Universal Robots PolyScope program: var_counter_106.urp

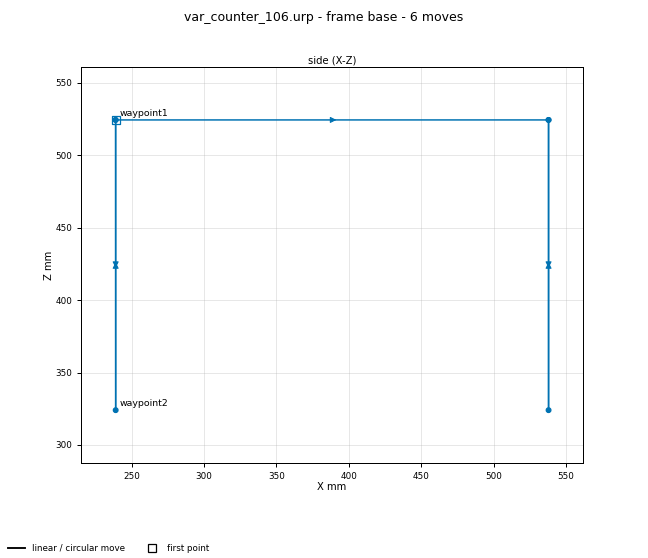
[picture p0: tool path of var_counter_106.urp in frame base, 6 of 6 moves have a stored position in this frame; points joined in program order, loops and branches not executed]
Program var_counter_106 (createdIn=3.2.19293 lastSavedIn=3.2.19293 directory=/programs installation=default robotSerialNumber=2015351391)
Calibrated DH parameters: a=[0.000352, -0.161198, -0.373486, 0.00005, 0.000049, 0]; d=[0.089268, 352.477598, -320.08558, -32.281492, 0.094939, 0.082518]; alpha=[1.570728, 0.001116, -0.003686, 1.571189, -1.570572, 0]; deltaTheta=[-0.000012, 1.181849, -1.491165, 0.309495, -0.000007, 0.000025]
Robot Program (runOnlyOnce=true motionType=MoveJ speed=1.047198 acceleration=1.396263 recalculateMotions=false)
  var_1 := 0
  Loop While (checkContinuously=false) expression=var_1<5
    Folder pick_part
      MoveL speed 250 mm/s, acceleration 1200 mm/s^2 (recalculateMotions=false) feature=Base
        Waypoint waypoint1: TCP in base x=238.987 y=198.778 z=524.462 mm, rx=-1.5848 ry=-0.1114 rz=-0.2808 rad; joints [52.485, -68.263, -119.544, 6.904, 121.33, -14.974] deg
        Waypoint waypoint2: TCP in base x=239.017 y=198.807 z=323.989 mm, rx=-1.585 ry=-0.1112 rz=-0.2807 rad; joints [52.411, -84.493, -141.527, 45.176, 121.522, -14.859] deg
        Set DigitalOutput pin=digital_out[4]; digitalValue=1
        Wait Sleep waitTime=0.5
        Waypoint waypoint1: TCP in base x=238.987 y=198.778 z=524.462 mm, rx=-1.5848 ry=-0.1114 rz=-0.2808 rad; joints [52.485, -68.263, -119.544, 6.904, 121.33, -14.974] deg
    Folder place_part
      MoveL speed 250 mm/s, acceleration 1200 mm/s^2 (recalculateMotions=false) feature=Base
        Waypoint waypoint3: TCP in base x=538.015 y=198.753 z=524.467 mm, rx=-1.5849 ry=-0.1113 rz=-0.2808 rad; joints [24.332, -109.201, -79.574, 7.141, 149.52, -15.82] deg
        Waypoint waypoint4: TCP in base x=538.025 y=198.76 z=323.991 mm, rx=-1.5849 ry=-0.1113 rz=-0.2808 rad; joints [24.308, -119.509, -96.212, 34.193, 149.628, -15.688] deg
        Set DigitalOutput pin=digital_out[4]; digitalValue=0
        Wait Sleep waitTime=0.5
        Waypoint waypoint3: TCP in base x=538.015 y=198.753 z=524.467 mm, rx=-1.5849 ry=-0.1113 rz=-0.2808 rad; joints [24.332, -109.201, -79.574, 7.141, 149.52, -15.82] deg
    var_1 := var_1+1
